SUBAPPLICATION Uebung_080c (* Beispiel für E_CTU mit Terminal-Ausgabe *)
  (* Standard: 61499-2; Description: Copyright (c) 2023 Meisterschulen am Ostbahnhof This program and the accompanying materials are made available under the terms of the Eclipse Public License 2.0 which is available at https://www.eclipse.org/legal/epl-2.0/ SPDX-License-Identifier: EPL-2.0 *)
  (* Version 1.1, 2026-04-21, Franz Höpfinger, Meisterschulen am Ostbahnhof, Added terminal output for counter value and restored logiBUS_IE *)
  PACKAGE Uebungen;
  IMPORT Uebungen::const::UT::DefaultPool::OutputNumber_N1;
  IMPORT logiBUS::io::DI::logiBUS_DI::Input_I1;
  IMPORT logiBUS::io::DI::logiBUS_DI::Input_I2;
  IMPORT logiBUS::io::DI::logiBUS_DI_Events::BUTTON_SINGLE_CLICK;
  IMPORT logiBUS::io::DQ::logiBUS_DO::Output_Q1;
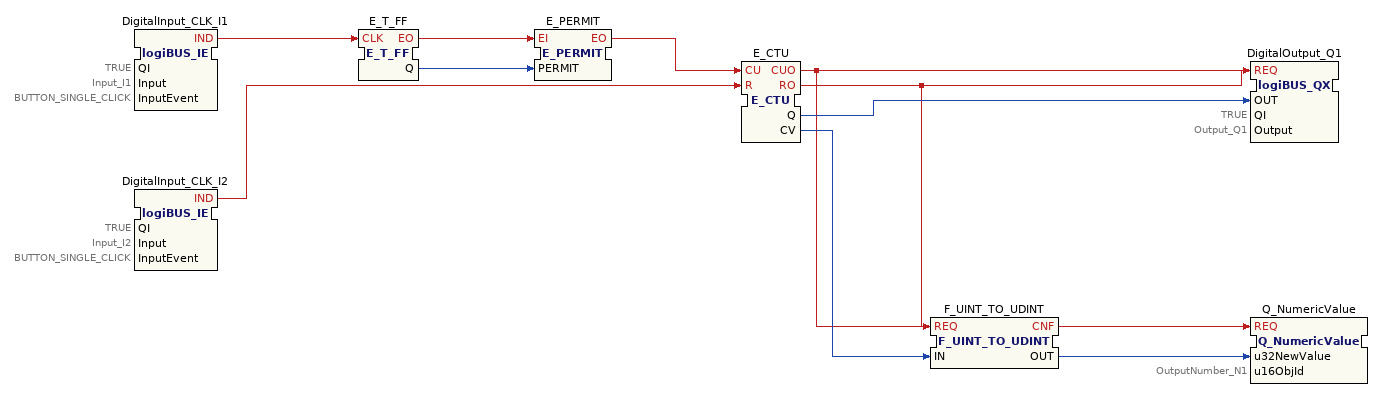
  FBS
    DigitalOutput_Q1 : logiBUS::io::DQ::logiBUS_QX(QI := TRUE, Output := Output_Q1);
    DigitalInput_CLK_I1 : logiBUS::io::DI::logiBUS_IE(QI := TRUE, Input := Input_I1, InputEvent := BUTTON_SINGLE_CLICK);
    E_CTU : iec61499::events::E_CTU;
    DigitalInput_CLK_I2 : logiBUS::io::DI::logiBUS_IE(QI := TRUE, Input := Input_I2, InputEvent := BUTTON_SINGLE_CLICK);
    E_PERMIT : iec61499::events::E_PERMIT;
    Q_NumericValue : isobus::UT::Q::Q_NumericValue(u16ObjId := OutputNumber_N1);
    F_UINT_TO_UDINT : iec61131::conversion::F_UINT_TO_UDINT;
    E_T_FF : iec61499::events::E_T_FF;
  END_FBS
  EVENT_CONNECTIONS
    DigitalInput_CLK_I1.IND TO E_T_FF.CLK;
    E_PERMIT.EO TO E_CTU.CU;
    DigitalInput_CLK_I2.IND TO E_CTU.R;
    E_CTU.CUO TO DigitalOutput_Q1.REQ;
    E_CTU.RO TO DigitalOutput_Q1.REQ;
    E_CTU.CUO TO F_UINT_TO_UDINT.REQ;
    E_CTU.RO TO F_UINT_TO_UDINT.REQ;
    F_UINT_TO_UDINT.CNF TO Q_NumericValue.REQ;
    E_T_FF.EO TO E_PERMIT.EI;
  END_CONNECTIONS
  DATA_CONNECTIONS
    E_CTU.Q TO DigitalOutput_Q1.OUT;
    E_CTU.CV TO F_UINT_TO_UDINT.IN;
    F_UINT_TO_UDINT.OUT TO Q_NumericValue.u32NewValue;
    E_T_FF.Q TO E_PERMIT.PERMIT;
  END_CONNECTIONS
END_SUBAPPLICATION
